{attribute 'qualified_only'}
VAR_GLOBAL
END_VAR

(* stored: Version 1.1.0.1, ProductVersion 3.1.4024.12
   GVL G_Outputs: Id {336e4417-bcc6-4cf5-be39-792bee9fdc47} *)
